FUNCTION_BLOCK FB_LamparaIntermitente_SFC
// La lampara parpadea de forma continua
VAR_INPUT
    TiempoParpadeo  : TIME := T#500MS;
END_VAR
VAR
    TiempoAnterior  : TIME;
    
    Lampara AT %Q*  : BOOL;
END_VAR

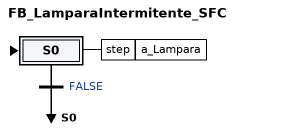
INITIAL_STEP S0:
    a_Lampara(N);  // step action
END_STEP
TRANSITION FROM S0 TO S0
    := FALSE;
END_TRANSITION

ACTION a_Lampara:
IF S0.t - TiempoAnterior > TiempoParpadeo THEN
    Lampara := NOT Lampara;
    TiempoAnterior := S0.t;
END_IF;
END_ACTION

END_FUNCTION_BLOCK

(* stored: Version 1.1.0.1, ProductVersion 3.1.4024.15
   POU FB_LamparaIntermitente_SFC: Id {ac299db4-ecb1-4502-977d-f799e68f966d}, SpecialFunc None
   Action a_Lampara: Id {eb69edbe-c575-4d2f-8b2f-5d305df408c8} *)
